// TIA Portal V20 export
VAR_GLOBAL   // PLC tag table "EROOM"
   cableReelDirectionFc7 AT %I225.3 : Bool;   // Cable reel Direction ("FC7")
   cableReelFeedingPointBypass AT %I225.4 : Bool;   // Cable reel Feeding point bypass Fast cam
   cableReelReelFull AT %I225.5 : Bool;   // Cable reel Reel full
   cableReelReferencePoint AT %I225.6 : Bool;   // Cable reel Reference point
   cableReelReelEmpty AT %I225.7 : Bool;   // Cable reel Reel empty
   cbRailClamp1 AT %I226.0 : Bool;   // Rail clamp 1 CB Feedback
   cbRailClamp1AntiCondHeating AT %I226.1 : Bool;   // Rail clamp 1 Anti-condensation heater CB Feedback
   cbRailClamp1CtrlCircuit AT %I226.2 : Bool;   // Rail clamp 1 control circuit CB Feedback
   railClamp1OilPumpContactorFb AT %I226.3 : Bool;   // Rail clamp 1 oil pump contactor Feedback
   railClamp1AntiCondHeatingContactorFb AT %I226.4 : Bool;   // Rail clamp 1 Anti-condensation heater contactor Feedback
   railClamp1LevelSw AT %I226.5 : Bool;   // Rail clamp 1 Level switch
   railClamp1TempSw AT %I226.6 : Bool;   // Rail clamp 1 Temperature switch
   "railClamp1LevelSw(1)" AT %I226.7 : Bool;   // Rail clamp 1 Level switch
   railClamp1BrakeReleased AT %I227.0 : Bool;   // Rail clamp 1 Brake released
   railLock1PosClosed AT %I227.2 : Bool;   // Rail lock 1 position Closed
   cbRailClamp2 AT %I228.0 : Bool;   // Rail clamp 2 CB Feedback
   cbRailClamp2AntiCondHeating AT %I228.1 : Bool;   // Rail clamp 2 Anti-condensation heater CB Feedback
   cbRailClamp2CtrlCircuit AT %I228.2 : Bool;   // Rail clamp 2 control circuit CB Feedback
   railClamp2OilPumpContactorFb AT %I228.3 : Bool;   // Rail clamp 2 oil pump contactor Feedback
   railClamp2AntiCondHeatingContactorFb AT %I228.4 : Bool;   // Rail clamp 2 Anti-condensation heater contactor Feedback
   railClamp2LevelSw AT %I228.5 : Bool;   // Rail clamp 2 Level switch
   railClamp2TempSw AT %I228.6 : Bool;   // Rail clamp 2 Temperature switch
   "railClamp2LevelSw(1)" AT %I228.7 : Bool;   // Rail clamp 2 Level switch
   railClamp2BrakeReleased AT %I229.0 : Bool;   // Rail clamp 2 Brake released
   railLock2PosClosed AT %I229.2 : Bool;   // Rail lock 2 position Closed
   cbERoomAc1Outdoor AT %I230.0 : Bool;   // E-Room A/C 1 outdoor unit CB Feedback
   cbERoomAc1Indoor AT %I230.1 : Bool;   // E-Room A/C 1 indoor unit CB Feedback
   cbERoomAc2Outdoor AT %I230.2 : Bool;   // E-Room A/C 2 outdoor unit CB Feedback
   cbERoomAc2Indoor AT %I230.3 : Bool;   // E-Room A/C 2 indoor unit CB Feedback
   cbERoomHeater AT %I230.4 : Bool;   // E-Room heater CB Feedback
   cbERoomHeaterCtrlCircuit AT %I230.5 : Bool;   // E-Room heater control circuit CB Feedback
   cbTrRoomCoolingFans AT %I231.0 : Bool;   // TR-Room cooling fans CB Feedback
   cbTrRoomHeater AT %I231.1 : Bool;   // TR-Room heater CB Feedback
   trRoomCoolingFansContactorFb AT %I231.2 : Bool;   // TR-Room cooling fans contactor Feedback
   trRoomHeaterContactorFb AT %I231.3 : Bool;   // TR-Room heater contactor Feedback
   cbTransformer400_230IllumSockets AT %I232.0 : Bool;   // 400/230V Illumination/ sockets transformer CB Feedback
   cbTransformer400_230 AT %I232.1 : Bool;   // 400/230V Transformer CB Feedback
   cbIllumPortalRcb AT %I232.2 : Bool;   // Illumination portal RCB Feedback
   cbIllumFloodlightsRcb AT %I232.3 : Bool;   // Illumination Floodlights RCB Feedback
   illumFloodlightsOnOffPb AT %I232.5 : Bool;   // Illumination Flood lights ON/OFF pushbutton
   cbIllumCableReelMaintPlatforms AT %I232.6 : Bool;   // Illumination Cable reel maintenance platforms CB Feedback
   cbSignalBeacons AT %I232.7 : Bool;   // Signal beacons CB Feedback
   cbC2_230VacSpare1 AT %I233.0 : Bool;   // +C2 230VAC spare CB Feedback
   cbC2_230VacSpare2 AT %I233.1 : Bool;   // +C2 230VAC spare CB Feedback
   cbIllumERoom AT %I234.0 : Bool;   // Illumination E-Room CB Feedback
   cbIllumTrRoom AT %I234.1 : Bool;   // Illumination TR-Room CB Feedback
   cbIllumMainStairs AT %I234.2 : Bool;   // Illumination Main stairsway CB Feedback
   cbIllumGirderNWE AT %I234.3 : Bool;   // Illumination Girder N, W and E sides CB Feedback
   cbIllumGirderWalkways AT %I234.4 : Bool;   // Illumination Girder main walkways CB Feedback
   cbIllumFestoonPlatforms AT %I234.5 : Bool;   // Illumination Festoon maintenance platforms CB Feedback
   cbIllumFloodLight1 AT %I234.6 : Bool;   // Illumination Flood light CB1 Feedback
   cbIllumFloodLight2 AT %I234.7 : Bool;   // Illumination Flood light CB2 Feedback
   cbIllumFloodLight3 AT %I235.0 : Bool;   // Illumination Flood light CB3 Feedback
   cbIllumFloodLight4 AT %I235.1 : Bool;   // Illumination Flood light CB4 Feedback
   illumFloodLight1ContactorFb AT %I235.2 : Bool;   // Illumination Flood light 1 contactor Feedback
   illumFloodLight2ContactorFb AT %I235.3 : Bool;   // Illumination Flood light 2 contactor Feedback
   illumFloodLight3ContactorFb AT %I235.4 : Bool;   // Illumination Flood light 3 contactor Feedback
   illumFloodLight4ContactorFb AT %I235.5 : Bool;   // Illumination Flood light 4 contactor Feedback
   swDoorERoomCtrlFb AT %I236.0 : Bool;   // E-Room door control switch Feedback
   swDoorTrRoomCtrlFb AT %I236.1 : Bool;   // TR-Room door control switch Feedback
   swFenceTrRoomCtrlFb AT %I236.2 : Bool;   // TR-Room fence control switch Feedback
   cabinEntranceInterlockContactorFb AT %I236.3 : Bool;   // Cabin entrance door interlock contactor Feedback
   craneEntranceGateAccessReq AT %I238.0 : Bool;   // Crane entrance gate Access request
   cabinEntranceGateAccessReq AT %I238.1 : Bool;   // Cabin entrance gate Access request
   cabinPlatformGateCtrlFb AT %I238.2 : Bool;   // Cabin platform gate control Feedback
   girderEntranceGateCtrlFb AT %I238.3 : Bool;   // Girder entrance gate control Feedback
   cabinEntranceInterlockMagnetPosNo AT %I238.4 : Bool;   // Cabin entrance interlock magnet position signaling contact (NO)
   lockOpenBtnGirderSide AT %I238.5 : Bool;   // Lock opening button girder side
   cbFireExtinguishingSystem AT %I238.6 : Bool;   // Fire extinguishing system CB Feedback
   fireExtinguishingSignal1 AT %I238.7 : Bool;   // Fire extinguishing system Signal 1
   fireExtinguishingSignal2 AT %I239.0 : Bool;   // Fire extinguishing system Signal 2
   fireExtinguishingSignal3 AT %I239.1 : Bool;   // Fire extinguishing system Signal 3
   fireExtinguishingSignal4 AT %I239.2 : Bool;   // Fire extinguishing system Signal 4
   fireExtinguishingSignal5 AT %I239.3 : Bool;   // Fire extinguishing system Signal 5
   fireExtinguishingSignal6 AT %I239.4 : Bool;   // Fire extinguishing system Signal 6
   fireExtinguishingSignal7 AT %I239.5 : Bool;   // Fire extinguishing system Signal 7
   mainCBSafetyRly AT %Q172.0 : Bool;   // Main CB Safety relay
   ltBrakeMC1Start AT %Q172.1 : Bool;   // LT brakes control Contactor 1
   ltBrakeMC2Start AT %Q172.2 : Bool;   // LT brakes control Contactor 2
   slSTO AT %Q172.3 : Bool;   // SL Motor module enable
   lt1STO AT %Q177.0 : Bool;   // LT1 Motor module enable
   lt2STO AT %Q177.1 : Bool;   // LT2 Motor module enable
   lt3STO AT %Q177.2 : Bool;   // LT3 Motor module enable
   lt4STO AT %Q177.3 : Bool;   // LT4 Motor module enable
   mh1STO AT %Q182.0 : Bool;   // MH1 Motor module enable
   mh2STO AT %Q182.1 : Bool;   // MH2 Motor module enable
   ct1STO AT %Q182.2 : Bool;   // CT1 Motor module enable
   ct2STO AT %Q182.3 : Bool;   // CT2 Motor module enable
   cabinEntranceInterlockStart AT %Q187.0 : Bool;   // Cabin entrance door interlock control
   signalBeaconTone1 AT %Q200.0 : Bool;   // Signal beacons tone C1 relay
   signalBeaconTone2 AT %Q200.1 : Bool;   // Signal beacons tone C2 relay
   illumMainStairwayStart AT %Q200.2 : Bool;   // Illumination Main stairsway ON/OFF (impulse control)
   illumEroomStart AT %Q200.3 : Bool;   // Illumination E-Room ON/OFF (impulse control)
   illumTrRoomStart AT %Q200.4 : Bool;   // Illumination TR-Room ON/OFF (impulse control)
   illumGirderFestoonStart AT %Q200.5 : Bool;   // Illumination Girder & Festoon maintenance platform ON/OFF (impulse control)
   illumFloodLight1Start AT %Q201.0 : Bool;   // Illumination Flood light group 1 ON/OFF (impulse control)
   illumFloodLight2Start AT %Q201.1 : Bool;   // Illumination Flood light group 2 ON/OFF (impulse control)
   illumFloodLight3Start AT %Q201.2 : Bool;   // Illumination Flood light group 3 ON/OFF (impulse control)
   illumFloodLightTruckStart AT %Q201.3 : Bool;   // Illumination Flood light Truck area ON/OFF (impulse control)
   illumCableReelStart AT %Q201.5 : Bool;   // Illumination Cable reel maintenance platform ON/OFF (impulse control)
   antiColWestOut1 AT %Q201.6 : Bool;   // LT anticollision system CU west side Input 1
   antiColWestOut2 AT %Q201.7 : Bool;   // LT anticollision system CU west side Input 2
   ltAntiCondHeatingMCStart AT %Q202.0 : Bool;   // LT Anti-condensation heating Contactor
   railClamp1PumpMCStart AT %Q202.1 : Bool;   // Rail clamp 1 oil pump contactor
   railClamp1HeaterMCStart AT %Q202.2 : Bool;   // Rail clamp 1Anti-condensation heater contactor
   railClamp1ValveStart AT %Q202.3 : Bool;   // Rail clamp 1 Valve control relay
   railClamp2PumpMCStart AT %Q202.4 : Bool;   // Rail clamp 2 oil pump contactor
   railClamp2HeaterMCStart AT %Q202.5 : Bool;   // Rail clamp 2 Anti-condensation heater contactor
   railClamp2ValveStart AT %Q202.6 : Bool;   // Rail clamp 2 Valve control relay
   eRoomAirCond1MCStart AT %Q203.4 : Bool;   // E-Room Air conditioner 1 Contactor
   eRoomAirCond2MCStart AT %Q203.5 : Bool;   // E-Room Air conditioner 2 Contactor
   antiColEastOut1 AT %Q203.6 : Bool;   // LT anticollision system CU east side Input 1
   antiColEastOut2 AT %Q203.7 : Bool;   // LT anticollision system CU east side Input 2
   iEroomTemp AT %IW240 : Int;   // E-Room temperature
   rlyEmStopRemoteCtrlCh2VS AT %I137.4 : Bool;   // Remote control Emergency Stop Channel 2 supply
   rlyStopRemoteCtrlCh1 AT %I136.1 : Bool;   // Remote control Stop Channel 1
   rlyEmStopRemoteCtrlCh1VS AT %I137.0 : Bool;   // Remote control Emergency Stop Channel 1 supply
   rlyEmStopRemoteCtrlCh2 AT %I136.4 : Bool;   // Remote control Emergency Stop Channel 2
   rlyStopRemoteCtrlCh2VS AT %I137.5 : Bool;   // Remote control Stop Channel 1 supply
   remoteCtrlST2 AT %I213.5 : Bool;   // Remote control ST2
   remoteCtrlST1 AT %I213.4 : Bool;   // Remote control ST1
   rlyStopRemoteCtrlCh2 AT %I136.5 : Bool;   // Remote control Stop Channel 1
   rlyStopRemoteCtrlCh1VS AT %I137.1 : Bool;   // Remote control Stop Channel 1 supply
   remoteCtrlK7 AT %I213.6 : Bool;   // Remote control K7
   rlyEmStopRemoteCtrlCh1 AT %I136.0 : Bool;   // Remote control Emergency Stop Channel 1
   cb24RemoteRadioRx AT %I207.6 : Bool;   // Remote radio control receiver 24VCD supply CB Feedback
   cb24Cu320 AT %I207.4 : Bool;   // CU320 24VCD supply CB Feedback
   btnEmStopGirderSESideCh1VS AT %I119.3 : Bool;   // Emergency stop Southeast side Girder Channel 1 Supply
   ltLimitSwitchSpeedLimitBLD AT %I148.5 : Bool;   // LT limit switch contacts end stop right
   btnEmStopSupportNESideCh1 AT %I118.0 : Bool;   // Emergency stop Northeast side Support Channel 1
   lt1SwDisconnector AT %I212.4 : Bool;   // LT1 Switch - disconnector Feedback
   cbAuxCircuitsVoltageCtrlRly AT %I201.2 : Bool;   // AUX circuits voltage control relay CB Feedback
   lt2MotorTempCtrl4 AT %I214.3 : Bool;   // LT2 motor 4 temperature control
   ct1BrakeRlyStartedVS AT %I143.6 : Bool;   // CT1 Brake switch relay Feedback Channel supply
   ups24VdcBatteryMode AT %I204.3 : Bool;   // 24VDC UPS Battery mode
   lt4MotorTempCtrl4 AT %I218.3 : Bool;   // LT4 motor 4 temperature control
   cbLt2Motor3 AT %I215.1 : Bool;   // LT2 Motor 3 CB Feedback
   ctLimitSwitchStopBLDCh1 AT %I160.1 : Bool;   // CT end stop backward switch Channel 1
   iAmbientTemp AT %IW242 : Int;   // Ambient temperature
   cb24Lt3MoMo AT %I206.7 : Bool;   // LT3 MoMo 24VDC supply CB Feedback
   ctOverHeaderSw1 AT %I223.2 : Bool;   // CT over the header 1 switch
   lt3BrakeRlyStartedVS AT %I143.2 : Bool;   // LT3 Brake switch relay Feedback Channel supply
   swGirderEntranceGateCtrlCh2VS AT %I131.5 : Bool;   // Girder entrance gate control Channel 2 supply
   antiColWestIn1 AT %I210.5 : Bool;   // LT anticollision system CU west side Output 1
   cbPowerMonitoring400V AT %I200.5 : Bool;   // Power monitoring device 400V CB Feedback
   cbLt4Motor3 AT %I219.1 : Bool;   // LT4 Motor 3 CB Feedback
   cbLt3Motor2 AT %I217.0 : Bool;   // LT3 Motor 2 CB Feedback
   btnEmStopGirderSESideCh1 AT %I118.3 : Bool;   // Emergency stop Southeast side Girder Channel 1
   cbPowerMonitoring230V AT %I200.6 : Bool;   // Power monitoring device 230V CB Feedback
   cbCableReel230VHeating AT %I224.4 : Bool;   // Cable reel 230V heating power supply CB Feedback
   cbPnSwitchSupply AT %I208.0 : Bool;   // PN switch supply CB Feedback
   cbCtSensorsSupply AT %I208.7 : Bool;   // CT sensors supply CB Feedback
   insulationMonitoringRly2 AT %I202.1 : Bool;   // Insulation monitoring Feedback relay 2
   cbLt2Motor4 AT %I215.2 : Bool;   // LT2 Motor 4 CB Feedback
   slewingSwDisconnectorFuseMon AT %I221.1 : Bool;   // Slewing Switch - disconnector Fuse monitoring
   btnEmStopCableReelCh2 AT %I100.6 : Bool;   // Cable reel Emergency Stop Channel 2
   cbLt1Motor1 AT %I212.7 : Bool;   // LT1 Motor 1 CB Feedback
   lt4MotorTempCtrl1 AT %I218.0 : Bool;   // LT4 motor 1 temperature control
   btnEmStopGirderSESideCh2 AT %I118.7 : Bool;   // Emergency stop Southeast side Girder Channel 2
   cbWeightMeasurementDisplay AT %I202.7 : Bool;   // Weight measurement display CB Feedback
   btnEmStopSupportNWSideCh2 AT %I112.6 : Bool;   // Emergency stop Northwest side Support Channel 2
   cbTrolley400V3Ph_NLoadsERoom AT %I202.6 : Bool;   // Trolley 400V+N loads CB (E-Room) Feedback
   cbAuxCircuitsMain AT %I201.1 : Bool;   // AUX circuits main CB Feedback
   cbCt1Motor1 AT %I222.1 : Bool;   // CT1 Motor 1 CB Feedback
   cbLt2Motor2 AT %I215.0 : Bool;   // LT2 Motor 2 CB Feedback
   ups24VdcOk AT %I204.4 : Bool;   // 24VDC UPS 24VDC OK
   ctLimitSwitchStopBLDCh2 AT %I160.5 : Bool;   // CT end stop backward switch Channel 2
   lt2MotorTempCtrl1 AT %I214.0 : Bool;   // LT2 motor 1 temperature control
   cb24Lt4MoMo AT %I207.0 : Bool;   // LT4 MoMo 24VDC supply CB Feedback
   cbIllumSocketsTrolleyERoom AT %I211.6 : Bool;   // Illumination/sockets trolley CB (E-Room) Feedback
   ltLimitSwitchStopBLD AT %I148.1 : Bool;   // LT limit switch contacts end stop left
   spareSafety1Ch2VS AT %I119.6 : Bool;   // Spare Channel 2 Supply
   cbMainS120 AT %I200.0 : Bool;   // Main S120 CB Feedback
   cbTelpher5t400V AT %I224.0 : Bool;   // Telpher 5t 400V supply CB Feedback
   ct1BrakeRlyStarted AT %I142.6 : Bool;   // CT1 Brake switch relay Feedback
   ctLimitSwitchStopFRUCh2 AT %I160.4 : Bool;   // CT end stop forward switch Channel 2
   cbInsulationCtrl230V AT %I202.3 : Bool;   // Insulation control relay 230V CB Feedback
   lt4SwDisconnectorFb AT %I218.4 : Bool;   // LT4 Switch - disconnector Feedback
   cbTransformer400_400 AT %I201.6 : Bool;   // 400/400V Transformer CB Feedback
   cb24Mh2MoMo AT %I206.4 : Bool;   // MH2 MoMo 24VDC supply CB Feedback
   btnEmStopCableReelGateCh2VS AT %I125.5 : Bool;   // Cable reel entrance gate E-Stop Channel 2 Supply
   btnEmStopEroomCh2VS AT %I113.4 : Bool;   // E-Room Emergency Stop pushbutton Channel 2 Supply
   btnEmStopGirderSWSideCh2VS AT %I119.5 : Bool;   // Emergency stop Southwest side Girder Channel 2 Supply
   ctLimitSwitchParkingPos AT %I160.2 : Bool;   // CT parking position switch
   insulationMonitoringRly1 AT %I202.0 : Bool;   // Insulation monitoring Feedback relay 1
   cbLt1Motor3 AT %I213.1 : Bool;   // LT1 Motor 3 CB Feedback
   lt2MotorTempCtrl3 AT %I214.2 : Bool;   // LT2 motor 3 temperature control
   ltBrakesMC2Started AT %I210.4 : Bool;   // LT brakes control Contactor 2 feedback
   fbSlewBrakeSwRlyVS AT %I137.3 : Bool;   // Slewing Brake switch relay Feedback Channel supply
   ups24VdcAlarm AT %I204.5 : Bool;   // 24VDC UPS Alarm
   cbAnticollisionEastHeating AT %I211.2 : Bool;   // LT anticollision system CU east side Enclosure heating CB Feedback
   btnEmStopCableReelCh1VS AT %I101.2 : Bool;   // Cable reel Emergency Stop Channel 1 Supply
   cbERoomHmi AT %I207.7 : Bool;   // E-Room HMI CB Feedback
   btnEmStopEroomCh1 AT %I112.0 : Bool;   // E-Room Emergency Stop pushbutton Channel 1
   lt3MotorTempCtrl1 AT %I216.0 : Bool;   // LT3 motor 1 temperature control
   cb24Lt1MoMo AT %I206.5 : Bool;   // LT1 MoMo 24VDC supply CB Feedback
   btnEmStopSupportNESideCh2 AT %I118.4 : Bool;   // Emergency stop Northeast side Support Channel 2
   cbLt3Motor3 AT %I217.1 : Bool;   // LT3 Motor 3 CB Feedback
   lt1MotorTempCtrl1 AT %I212.0 : Bool;   // LT1 motor 1 temperature control
   btnEmStopCabinEntrancePlatformCh1VS AT %I125.3 : Bool;   // Emergency stop Cabin entrance platform Channel 1 Supply
   ctLimitSwitchStopFRUVS AT %I161.0 : Bool;   // CT end stop forward switch Channel supply
   btnEmStopGirderNWSideCh2 AT %I112.5 : Bool;   // Emergency stop Northwest side Girder Channel 2
   ltLimitSwitchSpeedLimitFRU AT %I148.0 : Bool;   // LT limit switch contacts speed reduction right
   ctLimitSwitchSpeedLimitBLDVS AT %I161.6 : Bool;   // CT speed reduction backward Channel supply
   btnEmStopCableReelCh2VS AT %I101.6 : Bool;   // Cable reel Emergency Stop Channel 2 Supply
   cbCuEnclosuresHeating AT %I211.3 : Bool;   // CU-enclosures heating power supply CB Feedback
   btnEmStopCraneEntranceGateCh2VS AT %I125.4 : Bool;   // Crane entrance gate E-Stop Channel 2 Supply
   btnEmStopGirderSESideCh2VS AT %I119.7 : Bool;   // Emergency stop Southeast side Girder Channel 2 Supply
   indCraneGateAccessPermitted AT %Q203.1 : Bool;   // Crane entrance gate Access permitted (indication)
   cbLtSensorsSupply AT %I208.6 : Bool;   // LT sensors supply CB Feedback
   cbCableReel400VPower AT %I224.2 : Bool;   // Cable reel 400V power supply CB Feedback
   lt4BrakeRlyStartedVS AT %I143.3 : Bool;   // LT4 Brake switch relay Feedback Channel supply
   cbInsulationCtrl400V AT %I202.2 : Bool;   // Insulation control relay 400V CB Feedback
   eRoomHeaterContactorFb AT %I230.6 : Bool;   // E-Room heater contactor Feedback
   cb24Ct2MoMo AT %I207.2 : Bool;   // CT2 MoMo 24VDC supply CB Feedback
   lt1MotorTempCtrl2 AT %I212.1 : Bool;   // LT1 motor 2 temperature control
   spareSafety1Ch1VS AT %I119.2 : Bool;   // Spare Channel 1 Supply
   lt3MotorTempCtrl4 AT %I216.3 : Bool;   // LT3 motor 4 temperature control
   swFenceTrRoomCh2 AT %I106.6 : Bool;   // TR-Room fence control switch Channel 2
   auxCircuitsSwDisconnectorFuseMon AT %I201.0 : Bool;   // AUX circuits switch-disconnector Fuse monitoring
   btnEmStopSupportNESideCh2VS AT %I119.4 : Bool;   // Emergency stop Northeast side Support Channel 2 Supply
   swFenceTrRoomCh2VS AT %I107.6 : Bool;   // TR-Room fence control switch Channel 2 supply
   auxCircuitsChangeoverSwMainPos AT %I200.3 : Bool;   // Aux circuits changeover switch Main source position
   btnEmStopSupportNWSideCh1VS AT %I113.2 : Bool;   // Emergency stop Northwest side Support Channel 1 Supply
   btnEmStopCraneEntranceGateCh1VS AT %I125.0 : Bool;   // Crane entrance gate E-Stop Channel 1 Supply
   ups24VdcBatGt85 AT %I204.7 : Bool;   // 24VDC UPS BAT.>85%
   btnEmStopCableReelGateCh1 AT %I124.1 : Bool;   // Cable reel entrance gate E-Stop Channel 1
   ups24VdcReadyToBuffer AT %I204.6 : Bool;   // 24VDC UPS Ready to buffer
   cbCt2Motor1 AT %I222.6 : Bool;   // CT2 Motor 1 CB Feedback
   ctLimitSwitchSpeedLimitFRUVS AT %I161.3 : Bool;   // CT speed reduction forward Channel supply
   btnEmStopGirderNWSideCh2VS AT %I113.5 : Bool;   // Emergency stop Northwest side Girder Channel 2 Supply
   cbLtAntiCondHeating AT %I210.1 : Bool;   // LT Anti-condensation heating CB Feedback
   cbLt3MoMoFan AT %I216.5 : Bool;   // LT3 MoMo Fan CB Feedback
   lt2SwDisconnectorFb AT %I214.4 : Bool;   // LT2 Switch - disconnector Feedback
   mh2BrakeRlyStarted AT %I142.5 : Bool;   // Main Hoist 2 Brake switch relay
   cbLt4MoMoFan AT %I218.5 : Bool;   // LT4 MoMo Fan CB Feedback
   swCabinEntranceInterlockedCh1 AT %I106.3 : Bool;   // Cabin entrance interlock magnet position Channel 1
   cbAim230AC AT %I203.2 : Bool;   // AIM 230AC supply CB Feedback
   cbAlmFan AT %I203.3 : Bool;   // ALM Fan CB Feedback
   swCabinPlatformGateCtrlCh1VS AT %I131.0 : Bool;   // Cabin platform gate control Channel 1 supply
   cbMotorProtectionRelaysOpticTx AT %I208.5 : Bool;   // Motor protection relays, optic transmitters CB Feedback
   cb24VdcPs2 AT %I204.1 : Bool;   // 24VDC PS2 CB Feedback
   swDoorEroomCh1 AT %I106.0 : Bool;   // E-Room door control switch Channel 1
   ct2BrakeRlyStartedVS AT %I143.7 : Bool;   // CT2 Brake switch relay Feedback Channel supply
   lt2MotorTempCtrl2 AT %I214.1 : Bool;   // LT2 motor 2 temperature control
   btnEmStopGirderNESideCh1VS AT %I113.3 : Bool;   // Emergency stop Northeast side Girder Channel 1 Supply
   ps24VdcPs1Ok AT %I204.2 : Bool;   // 24VDC PS1 OK
   btnEmStopGirderSWSideCh2 AT %I118.5 : Bool;   // Emergency stop Southwest side Girder Channel 2
   ltLimitSwitchStopFRU AT %I148.4 : Bool;   // LT limit switch contacts speed reduction left
   cb24BrakingModule AT %I206.2 : Bool;   // Braking module 24VCD supply CB Feedback
   cableReelOvertensionMinusFc3 AT %I225.0 : Bool;   // Cable reel Overtension minus ("FC3")
   indCabinGateAccessRequest AT %Q203.2 : Bool;   // Cabin entrance gate Access request (indication)
   btnEmStopEroomCh2 AT %I112.4 : Bool;   // E-Room Emergency Stop pushbutton Channel 2
   cbSlewingMotor1 AT %I221.2 : Bool;   // Slewing Motor 1 CB Feedback
   cbCt2Motor2 AT %I222.7 : Bool;   // CT2 Motor 2 CB Feedback
   swFenceTrRoomCh1VS AT %I107.2 : Bool;   // TR-Room fence control switch Channel 1 supply
   mh1BrakeRlyStartedVS AT %I143.4 : Bool;   // Main Hoist 1 Brake switch relay Channel supply
   btnEmStopSupportNWSideCh1 AT %I112.2 : Bool;   // Emergency stop Northwest side Support Channel 1
   swCabinEntranceInterlockedCh2 AT %I106.7 : Bool;   // Cabin entrance interlock magnet position Channel 2
   cbTelephoneSystemSupply AT %I208.2 : Bool;   // Telephone system supply CB Feedback
   cbLt1MoMoFan AT %I212.5 : Bool;   // LT1 MoMo Fan CB Feedback
   swDoorEroomCh2 AT %I106.4 : Bool;   // E-Room door control switch Channel 2
   cbAnticollisionWestHeating AT %I210.7 : Bool;   // LT anticollision system CU west side Enclosure heating CB Feedback
   cbLt3Motor1 AT %I216.7 : Bool;   // LT3 Motor 1 CB Feedback
   cbMh2MoMoFan AT %I220.5 : Bool;   // MH2 MoMo Fan CB Feedback
   cbPanelPcSupply AT %I208.1 : Bool;   // Panel PC supply CB Feedback
   ctOverHeaderSw2 AT %I223.3 : Bool;   // CT over the header 2 switch
   mh1BrakeRlyStarted AT %I142.4 : Bool;   // Main Hoist 1 Brake switch relay
   ct1SwDisconnectorFb AT %I222.0 : Bool;   // CT1 Switch - disconnector Feedback
   cb24SlewingMoMo AT %I207.3 : Bool;   // Slewing MoMo 24VDC supply CB Feedback
   lt1Spare AT %I213.3 : Bool;   // LT1 Spare
   cbMainCtrlCircuits AT %I201.4 : Bool;   // Main CB control circuits CB Feedback
   spareSafety2Ch2VS AT %I125.6 : Bool;   // Spare Channel 2 Supply
   cb24Alm AT %I206.1 : Bool;   // ALM 24VCD supply CB Feedback
   btnEmStopCableReelCh1 AT %I100.2 : Bool;   // Cable reel Emergency Stop Channel 1
   cb24Lt2MoMo AT %I206.6 : Bool;   // LT2 MoMo 24VDC supply CB Feedback
   swDoorTrRoomCh1 AT %I106.1 : Bool;   // TR-Room door control switch Channel 1
   cbMh1MoMoFan AT %I220.1 : Bool;   // MH1 MoMo Fan CB Feedback
   btnEmStopSupportNESideCh1VS AT %I119.0 : Bool;   // Emergency stop Northeast side Support Channel 1 Supply
   cbLt2Motor1 AT %I214.7 : Bool;   // LT2 Motor 1 CB Feedback
   cbInterlocksSupply AT %I209.2 : Bool;   // Interlocks supply CB Feedback
   swGirderEntranceGateCtrlCh1VS AT %I131.1 : Bool;   // Girder entrance gate control Channel 1 supply
   swCabinPlatformGateCtrlCh2 AT %I130.4 : Bool;   // Cabin platform gate control Channel 2
   btnEmStopGirderSWSideCh1VS AT %I119.1 : Bool;   // Emergency stop Southwest side Girder Channel 1 Supply
   auxCircuitsChangeoverSwEmergencyPos AT %I200.4 : Bool;   // Aux circuits changeover switch Emergency source position
   lt1BrakeRlyStarted AT %I142.0 : Bool;   // LT1 Brake switch relay Feedback
   antiColEastIn2 AT %I211.1 : Bool;   // LT anticollision system CU east side Output 2
   cbTransformer400_400Secondary AT %I201.7 : Bool;   // 400/400V Transformer secondary CB Feedback
   btnEmStopSupportNWSideCh2VS AT %I113.6 : Bool;   // Emergency stop Northwest side Support Channel 2 Supply
   cb24Smc30DqHub AT %I207.5 : Bool;   // SMC30, DQ-hub 24VCD supply CB Feedback
   cbLt4Motor1 AT %I218.7 : Bool;   // LT4 Motor 1 CB Feedback
   ps24VdcPs2Ok AT %I205.0 : Bool;   // 24VDC PS2 OK
   ctLimitSwitchParkingPosVS AT %I161.2 : Bool;   // CT parking position switch Channel supply
   cb24Ct1MoMo AT %I207.1 : Bool;   // CT1 MoMo 24VDC supply CB Feedback
   btnEmStopGirderNESideCh2 AT %I112.7 : Bool;   // Emergency stop Northeast side Girder Channel 2
   lt4MotorTempCtrl3 AT %I218.2 : Bool;   // LT4 motor 3 temperature control
   swDoorEroomCh2VS AT %I107.4 : Bool;   // E-Room door control switch Channel 2 supply
   cableReelOvertensionPlusFc5 AT %I225.1 : Bool;   // Cable reel Overtension plus ("FC5")
   spareSafety1Ch1 AT %I118.2 : Bool;   // Spare Channel 1
   cbSensorsSupply AT %I209.1 : Bool;   // Sensors supply CB Feedback
   btnEmStopCableReelGateCh1VS AT %I125.1 : Bool;   // Cable reel entrance gate E-Stop Channel 1 Supply
   lt4BrakeRlyStarted AT %I142.3 : Bool;   // LT4 Brake switch relay Feedback
   cbCt1Motor2 AT %I222.2 : Bool;   // CT1 Motor 2 CB Feedback
   cbLt4Motor2 AT %I219.0 : Bool;   // LT4 Motor 2 CB Feedback
   surgeArrestersFb AT %I202.4 : Bool;   // Surge arresters Feedback
   swDoorEroomCh1VS AT %I107.0 : Bool;   // E-Room door control switch Channel 1 supply
   indCraneGateAccessRequest AT %Q203.0 : Bool;   // Crane entrance gate Access request (indication)
   ctOverHeaderSw4 AT %I223.5 : Bool;   // CT over the header 4 switch
   cableReelSlackDetectionFc6 AT %I225.2 : Bool;   // Cable reel Slack detection ("FC6")
   spareSafety1Ch2 AT %I118.6 : Bool;   // Spare Channel 2
   cbLtBrakes AT %I210.0 : Bool;   // LT Brakes CB Feedback
   cb24Aim AT %I206.0 : Bool;   // AIM 24VCD supply CB Feedback
   cbLt1Motor4 AT %I213.2 : Bool;   // LT1 Motor 4 CB Feedback
   cbEmergencySupplyVoltageCtrlRly AT %I201.3 : Bool;   // Emergency supply voltage control relay CB Feedback
   swDoorTrRoomCh2 AT %I106.5 : Bool;   // TR-Room door control switch Channel 2
   cbCraneEntranceMainCtrlCabinetHeaterERoom AT %I201.5 : Bool;   // Crane entrance main control cabinet heater CB (E-Room) Feedback
   antiColEastIn1 AT %I211.0 : Bool;   // LT anticollision system CU east side Output 1
   btnEmStopCraneEntranceGateCh1 AT %I124.0 : Bool;   // Crane entrance gate E-Stop Channel 1
   lt4MotorTempCtrl2 AT %I218.1 : Bool;   // LT4 motor 2 temperature control
   btnEmStopCableReelGateCh2 AT %I124.5 : Bool;   // Cable reel entrance gate E-Stop Channel 2
   spareSafety2Ch2 AT %I124.6 : Bool;   // Spare Channel 2
   cbSockets400VRCBO AT %I203.6 : Bool;   // Sockets 400V RCBO Feedback
   auxCircuitsVoltageCtrlRly AT %I200.1 : Bool;   // AUX circuits voltage control relay
   indCabinGateAccessPermitted AT %Q203.3 : Bool;   // Cabin entrance gate Access permitted (indication)
   slewBrakeRlyStarted AT %I136.3 : Bool;   // Slewing Brake switch relay Feedback
   swCabinPlatformGateCtrlCh1 AT %I130.0 : Bool;   // Cabin platform gate control Channel 1
   lt3MotorTempCtrl2 AT %I216.1 : Bool;   // LT3 motor 2 temperature control
   slewingSwDisconnectorFb AT %I221.0 : Bool;   // Slewing Switch - disconnector Feedback
   ctLimitSwitchStopFRUCh1 AT %I160.0 : Bool;   // CT end stop forward switch Channel 1
   ctLimitSwitchSpeedLimitFRU AT %I160.3 : Bool;   // CT speed reduction forward switch
   btnEmStopEroomCh1VS AT %I113.0 : Bool;   // E-Room Emergency Stop pushbutton Channel 1 Supply
   btnEmStopCabinEntrancePlatformCh2 AT %I124.7 : Bool;   // Emergency stop Cabin entrance platform Channel 2
   cbTrolley400VЗPhLoadsERoom AT %I202.5 : Bool;   // Trolley 400V loads CB (E-Room) Feedback
   lt3MotorTempCtrl3 AT %I216.2 : Bool;   // LT3 motor 3 temperature control
   ctOverHeaderSw3 AT %I223.4 : Bool;   // CT over the header 3 switch
   ct2SwDisconnectorFb AT %I222.5 : Bool;   // CT2 Switch - disconnector Feedback
   spareSafety2Ch1 AT %I124.2 : Bool;   // Spare Channel 1
   lt2BrakeRlyStarted AT %I142.1 : Bool;   // LT2 Brake switch relay Feedback
   cbInductiveSensorsSupply AT %I209.0 : Bool;   // Inductive sensors supply CB Feedback
   cbCableReel230VCtrl AT %I224.3 : Bool;   // Cable reel 230V control voltage power supply CB Feedback
   aimPrechargeSwDisconnectorFuseMon AT %I203.1 : Bool;   // AIM precharge switch-disconnector main contacts Fuse monitoring
   cbMotorHoursCounters24Vdc AT %I208.3 : Bool;   // Motor hours counters 24 VDC CB Feedback
   btnEmStopGirderSWSideCh1 AT %I118.1 : Bool;   // Emergency stop Southwest side Girder Channel 1
   auxCircuitsSwDisconnectorMainContactsFb AT %I200.7 : Bool;   // AUX circuits switch-disconnector main contacts Feedback
   btnEmStopGirderNWSideCh1 AT %I112.1 : Bool;   // Emergency stop Northwest side Girder Channel 1
   cbCraneEntranceMainCtrlCabinet AT %I209.3 : Bool;   // Crane entrance main control cabinet CB Feedback
   ctLimitSwitchStopBLDVS AT %I161.1 : Bool;   // CT end stop backward switch Channel supply
   btnEmStopCabinEntrancePlatformCh1 AT %I124.3 : Bool;   // Emergency stop Cabin entrance platform Channel 1
   swDoorTrRoomCh2VS AT %I107.5 : Bool;   // TR-Room door control switch Channel 2 supply
   mh1SwDisconnector AT %I220.0 : Bool;   // MH1 Switch - disconnector Feedback
   cbSlewingMotor2 AT %I221.3 : Bool;   // Slewing Motor 2 CB Feedback
   mh2BrakeRlyStartedVS AT %I143.5 : Bool;   // Main Hoist 2 Brake switch relay Channel supply
   surgeArrestersSwDisconnectorFuseMon AT %I203.5 : Bool;   // Surge arresters switch- disconnector Fuse monitoring
   cbSockets230VRCBO AT %I203.7 : Bool;   // Sockets 230V CB/RCB Feedback
   cbLt3Motor4 AT %I217.2 : Bool;   // LT3 Motor 4 CB Feedback
   swGirderEntranceGateCtrlCh1 AT %I130.1 : Bool;   // Girder entrance gate control Channel 1
   cb24Mh1MoMo AT %I206.3 : Bool;   // MH1 MoMo 24VDC supply CB Feedback
   ltAntiCondHeatingMCStarted AT %I210.2 : Bool;   // LT Anti-condensation heating contactor Feedback
   btnEmStopGirderNESideCh2VS AT %I113.7 : Bool;   // Emergency stop Northeast side Girder Channel 2 Supply
   ct2BrakeRlyStarted AT %I142.7 : Bool;   // CT2 Brake switch relay Feedback
   btnEmStopCabinEntrancePlatformCh2VS AT %I125.7 : Bool;   // Emergency stop Cabin entrance platform Channel 2 Supply
   lt1MotorTempCtrl3 AT %I212.2 : Bool;   // LT1 motor 3 temperature control
   cableReelHeatingFiberOk AT %I224.7 : Bool;   // Cable reel Heating fiber optic OK
   lt3SwDisconnectorFb AT %I216.4 : Bool;   // LT3 Switch - disconnector Feedback
   cbLt1Motor2 AT %I213.0 : Bool;   // LT1 Motor 2 CB Feedback
   cb24VdcPs1 AT %I204.0 : Bool;   // 24VDC PS1 CB Feedback
   aimPrechargeSwDisconnectorMainContactsFb AT %I203.0 : Bool;   // AIM precharge switch-disconnector main contacts Feedback
   emergencySupplyVoltageCtrlRly AT %I200.2 : Bool;   // Emergency supply voltage control relay
   swFenceTrRoomCh1 AT %I106.2 : Bool;   // TR-Room fence control switch Channel 1
   cb230VCircuitsTrolleyERoom AT %I211.7 : Bool;   // 230V circuits trolley CB (E-Room) Feedback
   lt2BrakeRlyStartedVS AT %I143.1 : Bool;   // LT2 Brake switch relay Feedback Channel supply
   btnEmStopGirderNWSideCh1VS AT %I113.1 : Bool;   // Emergency stop Northwest side Girder Channel 1 Supply
   btnEmStopCraneEntranceGateCh2 AT %I124.4 : Bool;   // Crane entrance gate E-Stop Channel 2
   cbAccessCircuits AT %I208.4 : Bool;   // Access circuits CB Feedback
   swDoorTrRoomCh1VS AT %I107.1 : Bool;   // TR-Room door control switch Channel 1 supply
   mh2SwDisconnector AT %I220.4 : Bool;   // MH2 Switch - disconnector Feedback
   spareSafety2Ch1VS AT %I125.2 : Bool;   // Spare Channel 1 Supply
   swGirderEntranceGateCtrlCh2 AT %I130.5 : Bool;   // Girder entrance gate control Channel 2
   cbLt4Motor4 AT %I219.2 : Bool;   // LT4 Motor 4 CB Feedback
   antiColWestIn2 AT %I210.6 : Bool;   // LT anticollision system CU west side Output 2
   ltBrakesMC1Started AT %I210.3 : Bool;   // LT brakes control Contactor 1 feedback
   btnEmStopGirderNESideCh1 AT %I112.3 : Bool;   // Emergency stop Northeast side Girder Channel 1
   surgeArrestersSwDisconnectorMainContactsFb AT %I203.4 : Bool;   // Surge arresters switch- disconnector main contacts Feedback
   lt1BrakeRlyStartedVS AT %I143.0 : Bool;   // LT1 Brake switch relay Feedback Channel supply
   lt3BrakeRlyStarted AT %I142.2 : Bool;   // LT3 Brake switch relay Feedback
   swCabinPlatformGateCtrlCh2VS AT %I131.4 : Bool;   // Cabin platform gate control Channel 2 supply
   ctLimitSwitchSpeedLimitBLD AT %I160.6 : Bool;   // CT speed reduction backward switch
   cbLt2MoMoFan AT %I214.5 : Bool;   // LT2 MoMo Fan CB Feedback
   lt1MotorTempCtrl4 AT %I212.3 : Bool;   // LT1 motor 4 temperature control
END_VAR
